% RSLogix 500 project P6_KOBIERSKI_M_v2.RSS, saved by version 8.30.00.16 %
PROJECT "UNTITLED"    % processor: Bul.1763 MicroLogix 1100 Series B %

PROGRAM FILES
  LAD 2 "MAIN"  10 rungs
  LAD 3 "COUNT"  1 rungs

DATA FILES
  O0 OUTPUT  4 elements
  I1 INPUT  6 elements
  S2 STATUS  66 elements
  B3 BINARY  1 elements
  T4 TIMER  4 elements
  C5 COUNTER  4 elements
  R6 CONTROL  1 elements
  N7 INTEGER  4 elements
  F8 FLOAT  1 elements

LADDER 2 "MAIN"
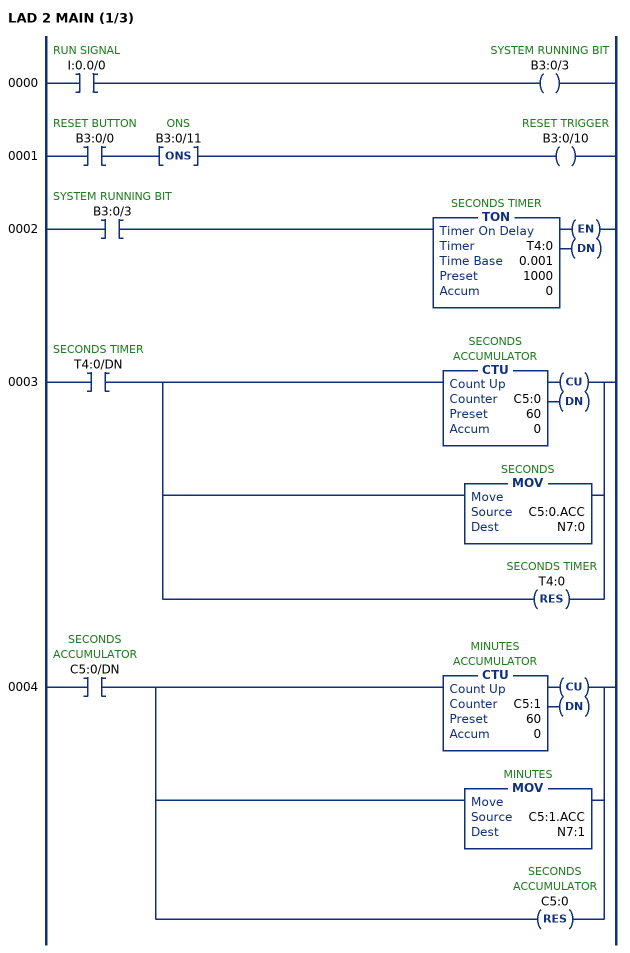
% Rung: 0 %
SOR XIC I:0.0/0 OTE B3:0/3 EOR
%   I:0.0/0  "RUN SIGNAL" %
%   B3:0/3  "SYSTEM RUNNING BIT" %
% Rung: 1 %
SOR XIC B3:0/0 ONS B3:0/11 OTE B3:0/10 EOR
%   B3:0/0  "RESET BUTTON" %
%   B3:0/11  "ONS" %
%   B3:0/10  "RESET TRIGGER" %
% Rung: 2 %
SOR XIC B3:0/3 TON T4:0 0.001 1000 0 EOR
%   B3:0/3  "SYSTEM RUNNING BIT" %
%   T4:0  "SECONDS TIMER" %
% Rung: 3 %
SOR XIC T4:0/DN BST CTU C5:0 60 0 NXB MOV C5:0.ACC N7:0 NXB RES T4:0 BND EOR
%   T4:0  "SECONDS TIMER" %
%   C5:0  "SECONDS ACCUMULATOR" %
%   N7:0  "SECONDS" %
% Rung: 4 %
SOR XIC C5:0/DN BST CTU C5:1 60 0 NXB MOV C5:1.ACC N7:1 NXB RES C5:0 BND EOR
%   C5:0  "SECONDS ACCUMULATOR" %
%   C5:1  "MINUTES ACCUMULATOR" %
%   N7:1  "MINUTES" %

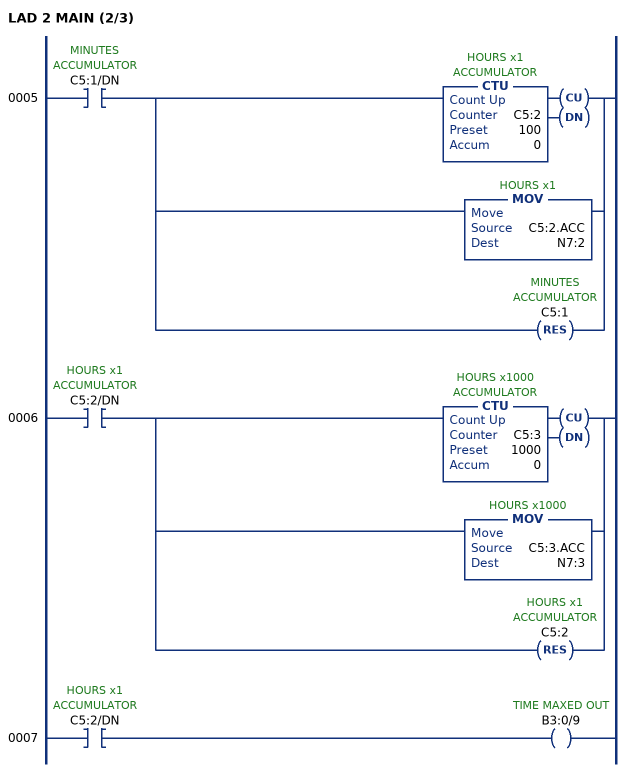
% Rung: 5 %
SOR XIC C5:1/DN BST CTU C5:2 100 0 NXB MOV C5:2.ACC N7:2 NXB RES C5:1 BND EOR
%   C5:1  "MINUTES ACCUMULATOR" %
%   C5:2  "HOURS x1 ACCUMULATOR" %
%   N7:2  "HOURS x1" %
% Rung: 6 %
SOR XIC C5:2/DN BST CTU C5:3 1000 0 NXB MOV C5:3.ACC N7:3 NXB RES C5:2 BND EOR
%   C5:2  "HOURS x1 ACCUMULATOR" %
%   C5:3  "HOURS x1000 ACCUMULATOR" %
%   N7:3  "HOURS x1000" %
% Rung: 7 %
SOR XIC C5:2/DN OTE B3:0/9 EOR
%   C5:2  "HOURS x1 ACCUMULATOR" %
%   B3:0/9  "TIME MAXED OUT" %

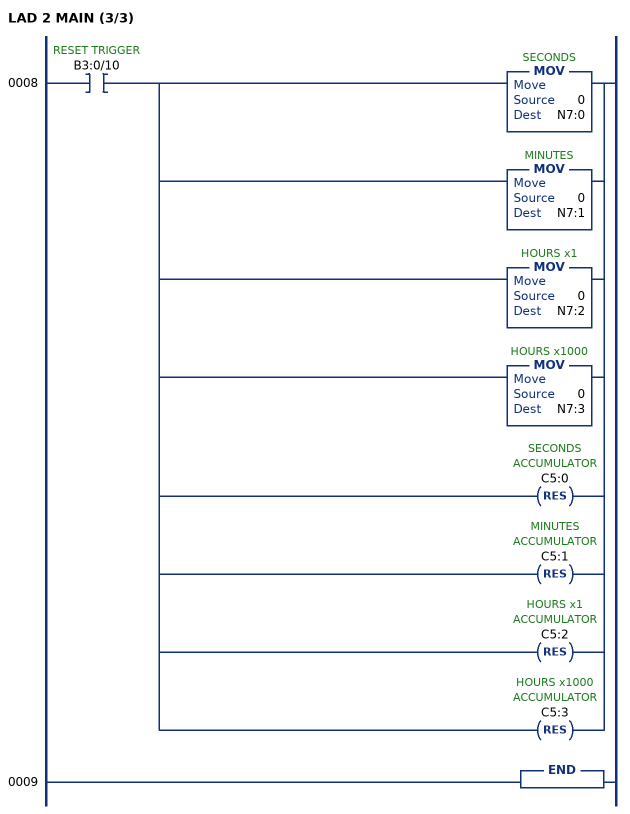
% Rung: 8 %
SOR XIC B3:0/10 BST MOV 0 N7:0 NXB MOV 0 N7:1 NXB MOV 0 N7:2 NXB MOV 0 N7:3 NXB RES C5:0 NXB RES C5:1 NXB RES C5:2 NXB RES C5:3 BND EOR
%   B3:0/10  "RESET TRIGGER" %
%   N7:0  "SECONDS" %
%   N7:1  "MINUTES" %
%   N7:2  "HOURS x1" %
%   N7:3  "HOURS x1000" %
%   C5:0  "SECONDS ACCUMULATOR" %
%   C5:1  "MINUTES ACCUMULATOR" %
%   C5:2  "HOURS x1 ACCUMULATOR" %
%   C5:3  "HOURS x1000 ACCUMULATOR" %
% Rung: 9 %
SOR END EOR

OTHER DOCUMENTED ADDRESSES
  B3:0/1  "ONS"
  B3:0/2  "TIMING RESET"
  B3:0/4  "ADD MINUTE"
  B3:0/5  "ONS"
  B3:0/6  "ONS"
  B3:0/7  "ADD HOUR"
  B3:0/8  "ADD HOUR x1000"
  U:3  "COUNT"

DATA TABLE (non-zero values as saved)
DATA T4
% .PRE .ACC %
% T4:0 % 1000 0
DATA C5
% .PRE .ACC %
% C5:0 % 60 0
% C5:1 % 60 0
% C5:2 % 100 0
% C5:3 % 1000 0
